# EPICS alarm handler configuration: apps/alhConfig/svtFlangeLV.alhConfig
#===============================================================================
# SVT Flange Board Low Voltage Config
#===============================================================================

GROUP NULL FLANGE_LV
$GUIDANCE
See SVT Ops manual sections relating to voltages.
PVs monitored by these alarms are supplied by the MPOD IOC (hvCaen).
$END

CHANNEL FLANGE_LV SVT:lv:fl:0:i_rd
$COMMAND  medm -x -attach -cmap -macro "sig=SVT:lv:fl:0:i_rd" aiaocalc_alarm.adl >> /dev/null
$GUIDANCE
The current supplied by this flange board low voltage channel has deviated from its normal value.
This usually indicates the channel is overloaded or disconnected, or that the hybrids have not yet been turned on.
Contact the SVT expert for further guidance.
$END

CHANNEL FLANGE_LV SVT:lv:fl:0:v_term
$COMMAND  medm -x -attach -cmap -macro "sig=SVT:lv:fl:0:v_term" aiaocalc_alarm.adl >> /dev/null
$GUIDANCE
The terminal voltage for this flange board low voltage channel has deviated from its normal value.
This usually indicates the channel is overloaded or disconnected.
Contact the SVT expert for further guidance.
$END

CHANNEL FLANGE_LV SVT:lv:fl:0:v_sens
$COMMAND  medm -x -attach -cmap -macro "sig=SVT:lv:fl:0:v_sens" aiaocalc_alarm.adl >> /dev/null
$GUIDANCE
The sense terminal voltage for this flange board low voltage channel has deviated from its nominal value of 5.5 V.
This usually indicates the channel is overloaded or disconnected.
Contact the SVT expert for further guidance.
$END

CHANNEL FLANGE_LV SVT:lv:fl:1:i_rd
$COMMAND  medm -x -attach -cmap -macro "sig=SVT:lv:fl:1:i_rd" aiaocalc_alarm.adl >> /dev/null
$GUIDANCE
The current supplied by this flange board low voltage channel has deviated from its normal value.
This usually indicates the channel is overloaded or disconnected, or that the hybrids have not yet been turned on.
Contact the SVT expert for further guidance.
$END

CHANNEL FLANGE_LV SVT:lv:fl:1:v_term
$COMMAND  medm -x -attach -cmap -macro "sig=SVT:lv:fl:1:v_term" aiaocalc_alarm.adl >> /dev/null
$GUIDANCE
The terminal voltage for this flange board low voltage channel has deviated from its normal value.
This usually indicates the channel is overloaded or disconnected.
Contact the SVT expert for further guidance.
$END

CHANNEL FLANGE_LV SVT:lv:fl:1:v_sens
$COMMAND  medm -x -attach -cmap -macro "sig=SVT:lv:fl:1:v_sens" aiaocalc_alarm.adl >> /dev/null
$GUIDANCE
The sense terminal voltage for this flange board low voltage channel has deviated from its nominal value of 5.5 V.
This usually indicates the channel is overloaded or disconnected.
Contact the SVT expert for further guidance.
$END

CHANNEL FLANGE_LV SVT:lv:fl:2:i_rd
$COMMAND  medm -x -attach -cmap -macro "sig=SVT:lv:fl:2:i_rd" aiaocalc_alarm.adl >> /dev/null
$GUIDANCE
The current supplied by this flange board low voltage channel has deviated from its normal value.
This usually indicates the channel is overloaded or disconnected, or that the hybrids have not yet been turned on.
Contact the SVT expert for further guidance.
$END

CHANNEL FLANGE_LV SVT:lv:fl:2:v_term
$COMMAND  medm -x -attach -cmap -macro "sig=SVT:lv:fl:2:v_term" aiaocalc_alarm.adl >> /dev/null
$GUIDANCE
The terminal voltage for this flange board low voltage channel has deviated from its normal value.
This usually indicates the channel is overloaded or disconnected.
Contact the SVT expert for further guidance.
$END

CHANNEL FLANGE_LV SVT:lv:fl:2:v_sens
$COMMAND  medm -x -attach -cmap -macro "sig=SVT:lv:fl:2:v_sens" aiaocalc_alarm.adl >> /dev/null
$GUIDANCE
The sense terminal voltage for this flange board low voltage channel has deviated from its nominal value of 5.5 V.
This usually indicates the channel is overloaded or disconnected.
Contact the SVT expert for further guidance.
$END

CHANNEL FLANGE_LV SVT:lv:fl:3:i_rd
$COMMAND  medm -x -attach -cmap -macro "sig=SVT:lv:fl:3:i_rd" aiaocalc_alarm.adl >> /dev/null
$GUIDANCE
The current supplied by this flange board low voltage channel has deviated from its normal value.
This usually indicates the channel is overloaded or disconnected, or that the hybrids have not yet been turned on.
Contact the SVT expert for further guidance.
$END

CHANNEL FLANGE_LV SVT:lv:fl:3:v_term
$COMMAND  medm -x -attach -cmap -macro "sig=SVT:lv:fl:3:v_term" aiaocalc_alarm.adl >> /dev/null
$GUIDANCE
The terminal voltage for this flange board low voltage channel has deviated from its normal value.
This usually indicates the channel is overloaded or disconnected.
Contact the SVT expert for further guidance.
$END

CHANNEL FLANGE_LV SVT:lv:fl:3:v_sens
$COMMAND  medm -x -attach -cmap -macro "sig=SVT:lv:fl:3:v_sens" aiaocalc_alarm.adl >> /dev/null
$GUIDANCE
The sense terminal voltage for this flange board low voltage channel has deviated from its nominal value of 5.5 V.
This usually indicates the channel is overloaded or disconnected.
Contact the SVT expert for further guidance.
$END
